FUNCTION_BLOCK HydraulicsIO EXTENDS SM_HydraulicsIO
VAR_INPUT
END_VAR
VAR_OUTPUT
END_VAR
VAR
END_VAR

SUPER^(safetyIO := safetyIO);

END_FUNCTION_BLOCK

(* stored: Version 1.1.0.1, ProductVersion 3.1.4018.5
   POU HydraulicsIO: Id {7d55bf3f-8cf9-4e3b-9df0-f3835bfa90dc}, SpecialFunc None *)
